// TIA Portal V17 export
// export: Created 2024-08-07T21:44:11.6686232Z, ExportSetting WithDefaults, DisplayName Totally Integrated Automation Portal, DisplayVersion V17 Update 7, DisplayName TIA Portal Openness, DisplayVersion V17 Update 7, DisplayName TIA Portal Version Control Interface, DisplayVersion V17, DisplayName SINAMICS Startdrive Advanced, DisplayVersion V17 SP2, DisplayName SINAMICS Startdrive G110M, G120, G120C, G120D, G120P, G115D, DisplayVersion V17 SP2, DisplayName SINAMICS Startdrive G130, G150, S120, S150, SINAMICS MV, S210, DisplayVersion V17 SP2, DisplayName STEP 7 Professional, DisplayVersion V17 Update 7, DisplayName STEP 7 Safety, DisplayVersion V17 Update 6, DisplayName WinCC Advanced / Unified PC, DisplayVersion V17 Update 7
DATA_BLOCK "MII_Interface_Configuration"   // DB2021
{ S7_Optimized_Access := 'TRUE' }
VERSION : 0.1
// stored: AutoNumber false, DBAccessibleFromOPCUA true, DBAccessibleFromWebserver true, IsOnlyStoredInLoadMemory false, IsRetainMemResEnabled false, IsWriteProtectedInAS false, MemoryReserve 100
   VAR
      Connection { ExternalAccessible := 'False'; ExternalVisible := 'False'; ExternalWritable := 'False'} : Struct
         ConnectInfo { ExternalAccessible := 'False'; ExternalVisible := 'False'; ExternalWritable := 'False'; S7_SetPoint := 'True'} : OPC_UA_SessionConnectInfo;
         ConnectionHdl { ExternalAccessible := 'False'; ExternalVisible := 'False'; ExternalWritable := 'False'} : DWord;
         ServerEndpointUrl { ExternalAccessible := 'False'; ExternalVisible := 'False'; ExternalWritable := 'False'} : String[254] := 'opc.tcp://:4840';
      END_STRUCT;
      Namespaces { ExternalAccessible := 'False'; ExternalVisible := 'False'; ExternalWritable := 'False'} : Struct
         NamespaceURIs { ExternalAccessible := 'False'; ExternalVisible := 'False'; ExternalWritable := 'False'} : Array[0..0] of WString;
         ServerNamespaceIndexes { ExternalAccessible := 'False'; ExternalVisible := 'False'; ExternalWritable := 'False'} : Array[0..0] of UInt;
         NamespaceStatusList { ExternalAccessible := 'False'; ExternalVisible := 'False'; ExternalWritable := 'False'} : Array[0..0] of DWord;
         NamespaceCount { ExternalAccessible := 'False'; ExternalVisible := 'False'; ExternalWritable := 'False'} : UInt := 1;
      END_STRUCT;
      MethodLists { ExternalAccessible := 'False'; ExternalVisible := 'False'; ExternalWritable := 'False'} : Struct
         MII_METHODS { ExternalAccessible := 'False'; ExternalVisible := 'False'; ExternalWritable := 'False'} : Struct
            MethodCount { ExternalAccessible := 'False'; ExternalVisible := 'False'; ExternalWritable := 'False'} : UInt := 9;
            ObjectNodes { ExternalAccessible := 'False'; ExternalVisible := 'False'; ExternalWritable := 'False'; S7_SetPoint := 'True'} : Array[0..8] of OPC_UA_NodeId;
            MethodNodes { ExternalAccessible := 'False'; ExternalVisible := 'False'; ExternalWritable := 'False'; S7_SetPoint := 'True'} : Array[0..8] of OPC_UA_NodeId;
            MethodHdls { ExternalAccessible := 'False'; ExternalVisible := 'False'; ExternalWritable := 'False'} : Array[0..8] of DWord;
         END_STRUCT;
      END_STRUCT;
   END_VAR
BEGIN
   Connection.ConnectInfo.SessionName := WSTRING#'OPC UA Connection_1';
   Connection.ConnectInfo.ApplicationName := WSTRING#'';
   Connection.ConnectInfo.SecurityMsgMode := 1;
   Connection.ConnectInfo.SecurityPolicy := 1;
   Connection.ConnectInfo.CheckServerCertificate := False;
   Connection.ConnectInfo.TransportProfile := 1;
   Connection.ConnectInfo.UserIdentityTokenType := 0;
   Connection.ConnectInfo.CertificateID := 0;
   Connection.ConnectInfo.SessionTimeout := T#30S;
   Connection.ConnectInfo.MonitorConnection := T#5S;
   Connection.ConnectInfo.LocaleIDs[0] := 'en-US';
   Connection.ConnectInfo.LocaleIDs[1..4] := '';
   Namespaces.NamespaceURIs[0] := WSTRING#'http://sap.com/PCoUaServer/Destinations';
   MethodLists.MII_METHODS.ObjectNodes[0..8].NamespaceIndex := 0;
   MethodLists.MII_METHODS.ObjectNodes[0..8].Identifier := WSTRING#'a72e725d-6be7-4a17-bcd4-0be67b6cbfbe';
   MethodLists.MII_METHODS.ObjectNodes[0..8].IdentifierType := 1;
   MethodLists.MII_METHODS.MethodNodes[0..8].NamespaceIndex := 0;
   MethodLists.MII_METHODS.MethodNodes[0].Identifier := WSTRING#'5e83d9d8-abe4-4ece-894f-119f40c23d1f';
   MethodLists.MII_METHODS.MethodNodes[1].Identifier := WSTRING#'3a6a30a3-a9b9-4f00-ac48-5dfb28f8e6a4';
   MethodLists.MII_METHODS.MethodNodes[2].Identifier := WSTRING#'fc62dbc1-f795-4566-bb4d-0b596c22b389';
   MethodLists.MII_METHODS.MethodNodes[3].Identifier := WSTRING#'c66a08a9-d6b4-453f-b0e9-0d4ff2f595c1';
   MethodLists.MII_METHODS.MethodNodes[4].Identifier := WSTRING#'a12cda35-f7c0-4943-b30d-d26694925508';
   MethodLists.MII_METHODS.MethodNodes[5].Identifier := WSTRING#'9febe458-2cc0-4c91-b17b-56067f98920d';
   MethodLists.MII_METHODS.MethodNodes[6].Identifier := WSTRING#'9fd0466f-1121-4821-944e-2d89fa189b19';
   MethodLists.MII_METHODS.MethodNodes[7].Identifier := WSTRING#'1a97343a-fec3-434f-bd32-25d77a49b705';
   MethodLists.MII_METHODS.MethodNodes[8].Identifier := WSTRING#'d0a2f4c1-2dea-442d-aa14-aa44dfe57828';
   MethodLists.MII_METHODS.MethodNodes[0..8].IdentifierType := 1;
END_DATA_BLOCK
